// TIA Portal V18 export
DATA_BLOCK "NoGoZoneV1_01_DB"   // DB86
VERSION : 0.1
// stored: AutoNumber true, DBAccessibleFromOPCUA true, InstanceOfName NoGoZoneV1, InstanceOfType FB
"NoGoZoneV1"
   // VAR_INPUT
   //    AutomateVersion : Int;
   //    MachineType : String;
   //    MachineLimit : Struct
   //       XSafety : Struct
   //          PosMax : DInt;
   //          PosMin : DInt;
   //          SafetyMargin : DInt;
   //          VelocityMax : DInt;
   //          VelocityMin : DInt;
   //       END_STRUCT;
   //       YSafety : Struct
   //          PosMax : DInt;
   //          PosMin : DInt;
   //          SafetyMargin : DInt;
   //          VelocityMax : DInt;
   //          VelocityMin : DInt;
   //       END_STRUCT;
   //       Z1Safety : Struct
   //          PosMax : DInt;
   //          PosMin : DInt;
   //          SafetyMargin : DInt;
   //          VelocityMax : DInt;
   //          VelocityMin : DInt;
   //       END_STRUCT;
   //       Z2Safety : Struct
   //          PosMax : DInt;
   //          PosMin : DInt;
   //          SafetyMargin : DInt;
   //          VelocityMax : DInt;
   //          VelocityMin : DInt;
   //       END_STRUCT;
   //       Heater : Struct
   //          FeedboxStart : DInt;
   //          FeedboxEnd : DInt;
   //          PrintboxStart : DInt;
   //          PrintboxEnd : DInt;
   //       END_STRUCT;
   //    END_STRUCT;
   //    XAxisHoming : Bool;
   //    YAxisHoming : Bool;
   //    Z1AxisHoming : Bool;
   //    Z2AxisHoming : Bool;
   //    ObjectHeight : DInt;
   //    ObjectWidth : DInt;
   //    ObjectMargin : DInt;
   //    ObjectActivate : Bool;
   //    XYstartendNormal : Struct
   //       XstartNormal : DInt;
   //       XendNormal : DInt;
   //       YstartNormal : DInt;
   //       YendNormal : DInt;
   //    END_STRUCT;
   //    XYstartendXL : Struct
   //       XstartXL : DInt;
   //       XendXL : DInt;
   //       YstartXL : DInt;
   //       YendXL : DInt;
   //    END_STRUCT;
   //    XActualPosition : DInt;
   //    YActualPosition : DInt;
   //    Z1ActualPosition : DInt;
   //    Z2ActualPosition : DInt;
   // END_VAR
   // VAR_OUTPUT
   //    NoGoAxisControl : Struct
   //       NoGoMotionLockXmove : Bool;
   //       NoGoMotionLockXjog : Bool;
   //       NoGoMotionLockYmove : Bool;
   //       NoGoMotionLockYjog : Bool;
   //       NoGoMotionLockZ1move : Bool;
   //       NoGoMotionLockZ1jog : Bool;
   //       NoGoMotionLockZ2move : Bool;
   //       NoGoMotionLockZ2jog : Bool;
   //       NoGoHomingPermissionX : Bool;
   //       NoGoHomingPermissionY : Bool;
   //       NoGoHomingPermissionZ1 : Bool;
   //       NoGoHomingPermissionZ2 : Bool;
   //       NoGoAlwaysMove : Bool;
   //    END_STRUCT;
   //    NoGoStatus : Struct
   //       NoGoZoneActive : Bool;
   //       YouAreInNoGoZoneWarning : Bool;
   //       NoGoZoneCollisionError : Bool;
   //    END_STRUCT;
   // END_VAR
   // VAR
   //    internalNoGoZoneXY : Struct
   //       internalNoGoZoneXstart : DInt;
   //       internalNoGoZoneXend : DInt;
   //       internalNoGoZoneYstart : DInt;
   //       internalNoGoZoneYend : DInt;
   //    END_STRUCT;
   //    internalNoGoZoneZ1start : DInt;
   //    internalNoGoZoneZ1end : DInt;
   //    internalNoGoZoneZ2start : DInt;
   //    internalNoGoZoneZ2end : DInt;
   //    internalObjectWithMargin : DInt;
   //    ControlCondition01 : Bool;
   //    ControlCondition02 : Bool;
   //    ControlCondition03 : Bool;
   // END_VAR
BEGIN
END_DATA_BLOCK
